PROGRAM STRAIGHTENING_PROG_1
VAR

	NEW: INT;
	FG: INT;
	ENABLE_TIMER: BOOL := FALSE;
	TMR1: TON;
	TMR2: TON;
	CNT1: CTU;
END_VAR

IF INPUT_VAR.STRAIGHTEN_START AND INDEXING_1_VAR.I_INDEXING_1_ROTATION_DONE THEN
	ENABLE_TIMER:=TRUE;
END_IF
IF ENABLE_TIMER THEN
	INPUT_VAR.STRAIGHTEN_START:=FALSE;
	TMR1(IN:=NOT TMR2.Q,PT:=T#0.15S);
	TMR2(IN:=TMR1.Q,PT:=T#0.3S);
	IF TMR2.Q THEN
		TMR1(IN:=FALSE); 
		TMR2(IN:=FALSE);
	END_IF
	
	(*IF NOT  INDEXING_1_VAR.I_PRESS_STOPPER_DOWN  THEN
		INDEXING_1_VAR.O_PRESS_STOPPER_DOWN:=TRUE;
		INDEXING_1_VAR.O_PRESS_STOPPER_UP:=FALSE;
	END_IF*)
ELSE
		TMR1(IN:=FALSE);
		TMR2(IN:=FALSE);
END_IF

CNT1(CU:=TMR1.Q,RESET:=NOT	ENABLE_TIMER,PV:=10);
//CNT1(CU:=TMR1.Q,RESET:=NOT INPUT_VAR.STRAIGHTEN_START,PV:=11);
IF CNT1.CV >=12 THEN
	ENABLE_TIMER:=FALSE;
	INDEXING_1_VAR.STRAIGHTEN_FINISH:=TRUE;
	INDEXING_1_VAR.O_PRESS_STOPPER_DOWN:=FALSE;
	INDEXING_1_VAR.O_PRESS_STOPPER_UP:=TRUE;
END_IF

IF CNT1.CV =2 THEN
	INDEXING_1_VAR.STRAIGHTEN_FINISH:=FALSE;
END_IF

IF 	INDEXING_1_VAR.STRAIGHTEN_FINISH THEN
	IF INDEXING_1_VAR.I_PRESS_STOPPER_UP THEN
		INPUT_VAR.STRAIGHTEN_DONE :=TRUE;	
		INPUT_VAR.STRAIGHTEN_PROCESS:=FALSE;
	END_IF	
END_IF
CASE CNT1.CV OF	
//CASE INDEXING_1_VAR.INDEXING_1_CASE OF
0:	
	INDEXING_1_VAR.O_PRESS_STOPPER_DOWN:=FALSE;
	INDEXING_1_VAR.O_PRESS_STOPPER_UP:=TRUE;
	INDEXING_1_VAR.I_INDEXING_1_READY_FOR_STRAIGHTEN:=FALSE;

1: 	INDEXING_1_VAR.O_PRESS_STOPPER_DOWN:=TRUE;
	INDEXING_1_VAR.O_PRESS_STOPPER_UP:=FALSE;

2: 	INDEXING_1_VAR.O_PRESS_STOPPER_DOWN:=TRUE;
	INDEXING_1_VAR.O_PRESS_STOPPER_UP:=FALSE;
	
3: 	INDEXING_1_VAR.O_PRESS_STOPPER_DOWN:=FALSE;
	INDEXING_1_VAR.O_PRESS_STOPPER_UP:=TRUE;
	
4: 	INDEXING_1_VAR.O_PRESS_STOPPER_DOWN:=TRUE;
	INDEXING_1_VAR.O_PRESS_STOPPER_UP:=FALSE;
5:	
	INPUT_VAR.STRAIGHTEN_PROCESS:=TRUE;
	INDEXING_1_VAR.O_INDEXING_1_GRIPPER_OPEN_1:=TRUE;
	INDEXING_1_VAR.O_INDEXING_1_GRIPPER_CLOSE_1:=FALSE;
		
6:
	INDEXING_1_VAR.O_INDEXING_1_GRIPPER_EXT_UP :=TRUE;	
	INDEXING_1_VAR.O_INDEXING_1_GRIPPER_EXT_down:=FALSE;
		
7:
	INDEXING_1_VAR.O_INDEXING_1_GRIPPER_OPEN_1:=FALSE;
	INDEXING_1_VAR.O_INDEXING_1_GRIPPER_CLOSE_1:=TRUE;
	//INDEXING_1_VAR.O_PRESS_STOPPER_DOWN:=FALSE;
	//INDEXING_1_VAR.O_PRESS_STOPPER_UP:=TRUE;		
8:
	INDEXING_1_VAR.O_INDEXING_1_GRIPPER_EXT_UP :=FALSE;	
	INDEXING_1_VAR.O_INDEXING_1_GRIPPER_EXT_down:=TRUE;
	
9:	
	INDEXING_1_VAR.O_INDEXING_1_GRIPPER_OPEN_1:=TRUE;
	INDEXING_1_VAR.O_INDEXING_1_GRIPPER_CLOSE_1:=FALSE;
	//INDEXING_1_VAR.O_PRESS_STOPPER_DOWN:=TRUE;
	//INDEXING_1_VAR.O_PRESS_STOPPER_UP:=FALSE;	
10:
	INDEXING_1_VAR.O_INDEXING_1_GRIPPER_EXT_UP :=TRUE;	
	INDEXING_1_VAR.O_INDEXING_1_GRIPPER_EXT_down:=FALSE;	
11:
	INDEXING_1_VAR.O_INDEXING_1_GRIPPER_OPEN_1:=FALSE;
	INDEXING_1_VAR.O_INDEXING_1_GRIPPER_CLOSE_1:=TRUE;
			
12:
	INDEXING_1_VAR.O_INDEXING_1_GRIPPER_EXT_UP :=FALSE;	
	INDEXING_1_VAR.O_INDEXING_1_GRIPPER_EXT_down:=TRUE;
	ENABLE_TIMER:=FALSE;
	INPUT_VAR.STRAIGHTEN_START:=FALSE;
END_CASE

IF 
	INDEXING_1_VAR.O_INDEXING_1_GRIPPER_OPEN_1 AND
	INDEXING_1_VAR.I_INDEXING_1_GRIPPER_OPEN_1 AND
	INDEXING_1_VAR.I_INDEXING_1_GRIPPER_OPEN_2	AND
	INDEXING_1_VAR.I_INDEXING_1_GRIPPER_OPEN_3	AND 
	INDEXING_1_VAR.I_INDEXING_1_GRIPPER_OPEN_4	AND
	NOT INDEXING_1_VAR.I_INDEXING_1_GRIPPER_CLOSE_1	AND
	NOT INDEXING_1_VAR.I_INDEXING_1_GRIPPER_CLOSE_2	AND
	NOT INDEXING_1_VAR.I_INDEXING_1_GRIPPER_CLOSE_3	AND
	NOT INDEXING_1_VAR.I_INDEXING_1_GRIPPER_CLOSE_4 THEN
		INDEXING_1_VAR.I_ALL_GRIPPER_OPEN :=TRUE;
	END_IF

IF 
	NOT INDEXING_1_VAR.O_INDEXING_1_GRIPPER_OPEN_1 AND
	NOT INDEXING_1_VAR.I_INDEXING_1_GRIPPER_OPEN_1 AND
	NOT INDEXING_1_VAR.I_INDEXING_1_GRIPPER_OPEN_2	AND
	NOT INDEXING_1_VAR.I_INDEXING_1_GRIPPER_OPEN_3	AND 
	NOT INDEXING_1_VAR.I_INDEXING_1_GRIPPER_OPEN_4	AND
	INDEXING_1_VAR.I_INDEXING_1_GRIPPER_CLOSE_1	AND
	INDEXING_1_VAR.I_INDEXING_1_GRIPPER_CLOSE_2	AND
	INDEXING_1_VAR.I_INDEXING_1_GRIPPER_CLOSE_3	AND
	INDEXING_1_VAR.I_INDEXING_1_GRIPPER_CLOSE_4 THEN
		INDEXING_1_VAR.I_ALL_GRIPPER_OPEN :=FALSE;
END_IF


	INDEXING_1_VAR.O_INDEXING_1_GRIPPER_OPEN_2:=INDEXING_1_VAR.O_INDEXING_1_GRIPPER_OPEN_1;
	INDEXING_1_VAR.O_INDEXING_1_GRIPPER_OPEN_3:=INDEXING_1_VAR.O_INDEXING_1_GRIPPER_OPEN_1;
	INDEXING_1_VAR.O_INDEXING_1_GRIPPER_OPEN_4:=INDEXING_1_VAR.O_INDEXING_1_GRIPPER_OPEN_1;

	INDEXING_1_VAR.O_INDEXING_1_GRIPPER_CLOSE_2:=INDEXING_1_VAR.O_INDEXING_1_GRIPPER_CLOSE_1;
	INDEXING_1_VAR.O_INDEXING_1_GRIPPER_CLOSE_3:=INDEXING_1_VAR.O_INDEXING_1_GRIPPER_CLOSE_1;
	INDEXING_1_VAR.O_INDEXING_1_GRIPPER_CLOSE_4:=INDEXING_1_VAR.O_INDEXING_1_GRIPPER_CLOSE_1;

END_PROGRAM

(* stored: Version 1.1.0.1, ProductVersion 3.1.4020.12
   POU STRAIGHTENING_PROG_1: Id {cd480fd6-f382-46f2-bea1-6edd10bfb24b}, SpecialFunc None *)
